// TIA Portal V19 export
VAR_GLOBAL   // PLC tag table "LB305"
   LB305_Scarico_Esterno_DX_Pb_ConfermaPaccoScaricato AT %I301.5 : Bool;   // 346SH3
   LB305_Scarico_Esterno_DX_Pb_Aux2 AT %I301.4 : Bool;   // 346SH2
   LB305_Scarico_Esterno_DX_Pb_PaccoReggiato AT %I301.3 : Bool;   // 346SH1
   LB305_Scarico_Esterno_DX_Lp_ConfermaPaccoScaricato AT %Q301.2 : Bool;   // 346SH3
   LB305_Scarico_Esterno_DX_Lp_Aux2 AT %Q301.1 : Bool;   // 346SH2
   LB305_Scarico_Esterno_DX_Lp_PaccoReggiato AT %Q301.0 : Bool;   // 346SH1
END_VAR
